Staubli VAL3: CloseFile.pgx

public program CloseFile()
begin


  //关闭所有文件
  call FileDir:CloseAllFile()
end
